FUNCTION_BLOCK FB_XTESFilterWheelCom
VAR_INPUT
	sCmd : STRING;
	bSend : BOOL;
END_VAR
VAR_IN_OUT
	(* 	I/O variables for a EL6001 terminal*)
	stIn_EL6001 : EL6inData22B;
	stOut_EL6001 : EL6outData22B;
END_VAR
VAR_OUTPUT
	sResponse : STRING;
	bDone : BOOL;
	eSerialLineErrorID : ComError_t;
	eSendErrorID : ComError_t;
	eRecvErrorID : ComError_t;
END_VAR
VAR
	// Communication Buffers
	TxBuffer : ComBuffer;
	RxBuffer : ComBuffer;
	fbClearComBuffer: ClearComBuffer;

	// Parameters for PLC -> EL6001
	fbEL6001Ctrl		: SerialLineControl;
	bEL6001CtrlError	: BOOL;
	eEL6001CtrlErrorID	: ComError_t;

	// Parameters for EL6001 -> FW
	Timer		: TON := (PT:=T#1S); (* time to pass before Q is set to TRUE *)
	fbSend		: SendString;
	bSendBusy	: BOOL;
	eLastSendErrorID: ComError_t;
	fbReceive		: ReceiveString;
	sReceivedString	: STRING;
	sLastReceivedString: STRING;
	bStringReceived	: BOOL;
	bReceiveBusy	: BOOL;
	bReceiveError	: BOOL;
	eReceiveErrorID	: ComError_t;
	bReceiveTimeout	: BOOL;
	nReceiveCounter	: UDINT;
	nSendCounter : UDINT;
	sStringToSend : STRING;

	fbFormatString : FB_FormatString;

	// Parameters for state-machine implementation
	nStep : INT := 0;
END_VAR

// Start Communicating with EL6001
fbEL6001Ctrl(
	Mode:= SERIALLINEMODE_EL6_22B, 
	pComIn:= ADR(stIn_EL6001), 
	pComOut:= ADR(stOut_EL6001), 
	SizeComIn:= SIZEOF(stIn_EL6001), 
	Error=> , 
	ErrorID=> eSerialLineErrorID, 
	TxBuffer:= TxBuffer, 
	RxBuffer:= RxBuffer );
IF fbEL6001Ctrl.Error THEN
	bEL6001CtrlError := TRUE;
	eEL6001CtrlErrorID := fbEL6001Ctrl.ErrorID;
END_IF

IF bSend THEN
	nStep := 10;
	bSend := FALSE;
	bDone := FALSE;
END_IF

// Attempt at solution that sends one command at a time, not on constant loop
CASE nStep OF
	0:
		; // idle
	10:
		// Clear buffers in case any lingering data
		fbClearComBuffer(Buffer:=TxBuffer);
		fbClearComBuffer(Buffer:=RxBuffer);
		// Prepare string to send
		sStringToSend := CONCAT(sCmd, '$R');
		// Send string
		fbSend(	SendString:= sStringToSend,
				TXbuffer:= TxBuffer,
				Busy=> bSendBusy,
				Error=> eSendErrorID);
		IF fbSend.Error <> COMERROR_NOERROR THEN
			eLastSendErrorID := fbSend.Error;
		ELSE
			nSendCounter := nSendCounter + 1;
		END_IF
		nStep := nStep + 10;
	20:
		// Finish sending String
		IF fbSend.Busy THEN
			fbSend(	SendString:= sStringToSend,
					TXbuffer:= TxBuffer,
					Busy=> bSendBusy,
					Error=> eSendErrorID);
			IF fbSend.Error <> COMERROR_NOERROR THEN
				eLastSendErrorID := fbSend.Error;
			ELSE
				nSendCounter := nSendCounter + 1;
			END_IF
		ELSE
			nStep := nStep + 10;
		END_IF
	30:
		// Get Reply
		fbReceive(
			Prefix:= '',
			Suffix:= '$R',
			Timeout:= T#100MS,
			ReceivedString:= sReceivedString,
			RXbuffer:= RxBuffer,
			StringReceived=> bStringReceived,
			Busy=> bReceiveBusy,
			Error=> eRecvErrorID,
			RxTimeout=> bReceiveTimeout );
		IF fbReceive.Error <> COMERROR_NOERROR THEN
			eReceiveErrorID := fbReceive.Error;
		END_IF

		IF bStringReceived THEN
			nReceiveCounter := nReceiveCounter + 1;
			// Check for response
			IF FIND(sReceivedString, sStringToSend)=0 THEN
				sResponse := sReceivedString;
				bDone := TRUE;
				nStep := 0;
			END_IF
		END_IF
END_CASE

END_FUNCTION_BLOCK

(* stored: Version 1.1.0.1, ProductVersion 3.1.4020.14
   POU FB_XTESFilterWheelCom: Id {1709bd62-5b3d-48ab-a1a1-083fae30a95e}, SpecialFunc None *)
